PROGRAM prgComEffIO
VAR
	fbCom		: FB_MqttCommunicator_V5;
	
	bHBTimmer: BOOL;							//{#lynus.ag#()}
	bHBSending: BOOL;							//{#lynus.ag#()}
	bError: BOOL;								//{#lynus.ag#()}
//	intTimerHB: DINT;							//{#lynus.ag#()}
	f_Trig_HB: f_trig;
	stringArray_Last_HB: ARRAY[0..50] OF STRING(30);
	intCount: INT;
	time_Temp: TIME;
END_VAR

fbCom(
	bConnect:= TRUE, 
	strAuthkey := 'ENE87365342998',
	sUserName:= 'e6a81f80-1adc-41aa-92f3-882fd2685fc6', 
	sUserPassword:= 'c755b11c-3f9d-40f0-ac27-e35cd683b09b', 
	eSavePositionCertificate:= eSavePositionOnPLC.ePostionC, 
	time_HeartBeat_sec := T#1S,
	bConnected=> , 
	bError=> , 
	hrErrorCode=> , 
	eConnectionState=> , 
	eErrorMessage_Out=> );
	
bHBTimmer 	:= fbCom.fbTimerHB.Q;
bHBSending 	:= fbCom.bHBSending;
bError		:= fbCom.bError;
// intTimerHB 	:= TIME_TO_DINT(fbCom.fbTimerHB.ET);

prg_SystemTime();
f_Trig_HB(CLK :=  fbCom.bHBSending);
IF f_Trig_HB.Q THEN
	IF intCount>50 OR intCount<0 THEN
		intCount:=0;
	END_IF
	stringArray_Last_HB[intCount] := prg_SystemTime.stringSystemTime_ms;
	intCount := intCount+1;
END_IF

time_Temp := fbCom.fbTimerHB.ET;

END_PROGRAM

(* stored: Version 1.1.0.1, ProductVersion 3.1.4024.13
   POU prgComEffIO: Id {cbcd318b-bf51-484c-bcaa-d6efcdf43fe3}, SpecialFunc None *)
